FUNCTION_BLOCK FB_MGMT_ThNTZ
VAR_INPUT
END_VAR
VAR_OUTPUT
END_VAR
VAR
	System_Waermetauscher_915				: FB_MGMT_ThNTZ_Aktor;
END_VAR

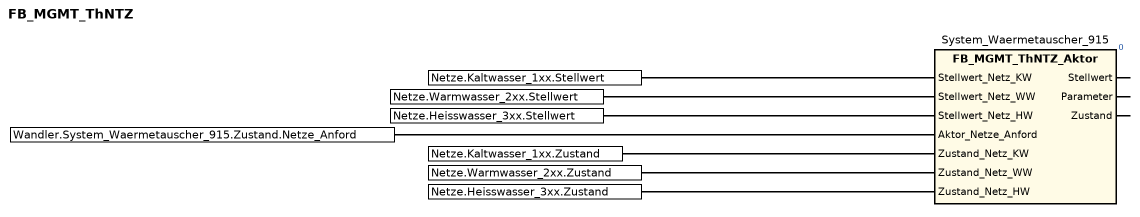
System_Waermetauscher_915(
    Stellwert_Netz_KW := Netze.Kaltwasser_1xx.Stellwert,
    Stellwert_Netz_WW := Netze.Warmwasser_2xx.Stellwert,
    Stellwert_Netz_HW := Netze.Heisswasser_3xx.Stellwert,
    Aktor_Netze_Anford := Wandler.System_Waermetauscher_915.Zustand.Netze_Anford,
    Zustand_Netz_KW := Netze.Kaltwasser_1xx.Zustand,
    Zustand_Netz_WW := Netze.Warmwasser_2xx.Zustand,
    Zustand_Netz_HW := Netze.Heisswasser_3xx.Zustand); // FB_MGMT_ThNTZ_Aktor

END_FUNCTION_BLOCK

(* stored: Version 1.1.0.1, ProductVersion 3.1.4024.9
   POU FB_MGMT_ThNTZ: Id {3aea63e1-c40c-4c28-9a62-394fe3829fc4}, SpecialFunc None *)
